{attribute 'GeneratedUsingTerminal: EJ2522-0000-0022'}
{attribute addProperty BoxType "EJ2522-0000-0022"}
{attribute addProperty Id "ControlAT %Q*Control_DAEE1D523Frequency_valueAT %Q*UINT2"}
{attribute addProperty CRC "2458384612"}
{attribute addProperty Size "5"}
TYPE PTO_Control_Channel_9287F8E4 :
STRUCT
	{attribute addProperty Name "Control"}
	Control AT %Q* : Control_DAEE1D52;
	{attribute addProperty Name "Frequency_value"}
	Frequency_value AT %Q* : UINT;
END_STRUCT
END_TYPE

(* stored: Version 1.2.0.0, ProductVersion 3.1.4024.9
   DUT PTO_Control_Channel_9287F8E4: Id {609a5568-e672-4e8b-9122-20ad74f60efb} *)
